// TwinCAT 3 PLC project Untitled1
// ProgramVersion: 3.1.4023.0
// libraries:
//   Tc2_Standard, * (Beckhoff Automation GmbH)
//   Tc2_System, * (Beckhoff Automation GmbH)
//   Tc3_Module, * (Beckhoff Automation GmbH)
// project tree:
//   / PlcTask.TcTTO (not stored), POU.TcPOU
//   POUs/ DUT.TcDUT, FB_Test.TcPOU, MAIN.TcPOU

// ---- POUs/DUT.TcDUT
TYPE DUT :
STRUCT
	v : BOOL;
END_STRUCT
END_TYPE

// ---- POU.TcPOU
FUNCTION_BLOCK POU
VAR_INPUT
END_VAR
VAR_OUTPUT
END_VAR
VAR
END_VAR

END_FUNCTION_BLOCK

// ---- POUs/FB_Test.TcPOU
FUNCTION_BLOCK FB_Test
VAR_INPUT
T	:BOOL;;
END_VAR
VAR_OUTPUT
END_VAR
VAR
END_VAR

T	:=TRUE;
//

END_FUNCTION_BLOCK

// ---- POUs/MAIN.TcPOU
PROGRAM MAIN
VAR
	
	X	:	INT;

END_VAR

x;//ujdff
// commentüüüü

END_PROGRAM
